Staubli VAL3: sendStatus.pgx

public program sendStatus()
  local num l_nRetVal
begin
  call sendData(siTcpIpFbk,rosStatusMsg.prefix.nData,nOutConnFlag)
  call sendData(siTcpIpFbk,rosStatusMsg.header.nData,nOutConnFlag)
  call sendData(siTcpIpFbk,rosStatusMsg.body.nData,nOutConnFlag)
end
